// TIA Portal V19 export
DATA_BLOCK "A0302_PareggiatoreTesta_PERS"   // DB123
// stored: MemoryReserve 100
   VAR RETAIN
      Par : Struct
         Ax : "Positioning_DOL_Machine_Par";
         Ax_Pers { ExternalAccessible := 'False'; ExternalVisible := 'False'; ExternalWritable := 'False'} : "Positioning_DOL_Machine_Pers_Data";
         Enc : "PosFbk_RTN";
         Ax_Aut : "A0301_Mach_Speed_Par";
         Bloccaggio_Sens : Struct
            "2111B1" : "Analogic_SensorManagement_Par";
            SogliaWork : Real := 0.0;
         END_STRUCT;
         CarroPareggTesta { ExternalAccessible := 'False'; ExternalVisible := 'False'; ExternalWritable := 'False'} : Struct
            Delay_StartMove : Time := T#100MS;
            Preset : LReal := 348.5;
         END_STRUCT;
         Cremaliera { ExternalAccessible := 'False'; ExternalVisible := 'False'; ExternalWritable := 'False'} : Struct
            Modulo : LReal := 2.5;
            Passo : LReal := 7.854;
         END_STRUCT;
      END_STRUCT;
      IEC_SP : Struct
         FTC_Rall : Struct
            TON_PT : Time := T#1MS;
            TOF_PT : Time := T#200MS;
         END_STRUCT;
         FTC_ProxLs : Struct
            TON_PT : Time := T#1MS;
            TOF_PT : Time := T#200MS;
         END_STRUCT;
         FTC_PresentMat : Struct
            TON_PT : Time := T#500MS;
            TOF_PT : Time := T#500MS;
         END_STRUCT;
         Check_2111B1 : Struct
            TON_PT : Time := T#500MS;
         END_STRUCT;
      END_STRUCT;
   END_VAR
BEGIN
   Par.Ax.PosTolerance := 0.5;
   Par.Ax.Minus_Limit := 338.5;
   Par.Ax.Plus_Limit := 2770.0;
   Par.Ax.PreCutOff := 0.2;
   Par.Ax.PreEndLowSpeed := 2.0;
   Par.Ax.PreEndMedSpeed := 5.0;
   Par.Ax.LowSpeed := 5.0;
   Par.Ax.MedSpeed := 10.0;
   Par.Ax.HighSpeed := 70.0;
   Par.Ax.Man_Speed := 20.0;
   Par.Ax_Pers.AxisHomed := TRUE;
   Par.Enc.Preset.Pulses := 402_167_584;
   Par.Enc.Preset.Units := 348.56;
   Par.Enc.Config.Resolution := -125.663706143592;
   Par.Ax_Aut.SemiAut_Vel := 50.0;
   Par.Ax_Aut.Aut_Vel := 50.0;
   Par.Ax_Aut.Aut_Acc := 1.0;
   Par.Ax_Aut.Aut_Dec := 1.0;
   Par.Bloccaggio_Sens."2111B1".Enable := TRUE;
   Par.Bloccaggio_Sens."2111B1".RangeLow := 0.0;
   Par.Bloccaggio_Sens."2111B1".RangeHigh := 0.0;
END_DATA_BLOCK
